// Mitsubishi GX Works2 project: Group555   PLC: FX3G

// global labels: Global1
VAR_GLOBAL
  StartDay AT X007 : BOOL;
  EmergencySwitch AT X011 : BOOL;
  StartLamp AT Y007 : BOOL;
  Yeast_start_register AT D1100 : REAL;
  Malt_start_register AT D1102 : REAL;
  Hops_start_register AT D1104 : REAL;
  Yeast_storage AT D1106 : REAL;
  Malt_storage AT D1108 : REAL;
  Hops_storage AT D1110 : REAL;
  update_storage AT M1 : BOOL;
  Start_cooking AT X001 : BOOL;
  analogInput AT D8280 : INT;
END_VAR
VAR_GLOBAL CONSTANT
  lagerLow : INT;
  PilsnerLow : INT := 2400;
  lager_top : INT := 2000;
  PilsnerTop : INT := 4000;
END_VAR
VAR_GLOBAL
  LagerChoosen AT M2 : BOOL;
  PilsnerChoosen AT M3 : BOOL;
END_VAR
VAR_GLOBAL CONSTANT
  MinYeasteLager : REAL := 150;
  MinMaltLager : REAL := 12;
  MinHopsLager : REAL := 60;
END_VAR
VAR_GLOBAL
  lagerCheackStorage AT M4 : BOOL;
  pilsnerCheackStorage AT M5 : BOOL;
END_VAR
VAR_GLOBAL CONSTANT
  timeLight : INT := 40;
END_VAR
VAR_GLOBAL
  TimerLightTS1 AT TS1 : BOOL;
  light AT Y001 : BOOL;
END_VAR
VAR_GLOBAL CONSTANT
  MinYeastePilsner : REAL := 120;
  MinMaltPilsner : REAL := 6;
  decYeastStorage : REAL := 150;
  decMoltStorage : REAL := 12;
  decHopsStorage : REAL := 60;
  decYeastStorage1 : REAL := 120;
  decMoltStorage1 : REAL := 6;
  decHopsStorage1 : REAL := 53;
END_VAR
VAR_GLOBAL
  Fermentation AT X005 : BOOL;
  FermentationLagerTimer AT TC2 : BOOL;
  TimerFlashLight1 AT TS2 : BOOL;
  light3 AT Y003 : BOOL;
  FermentatioPilnserrTimer AT TC3 : BOOL;
  FermentationLagerOverTimer AT TS2 : BOOL;
  FermentationPlisnerOverTimer AT TS3 : BOOL;
  TimerFermentationOver AT M6 : BOOL;
  Flasing AT X005 : BOOL;
  FlasingFake AT M7 : BOOL;
  FlasingTimer AT TC4 : BOOL;
END_VAR
VAR_GLOBAL CONSTANT
  Flashingtime : INT := 3;
END_VAR
VAR_GLOBAL
  FlashingTimer : INT;
  FlahingTimer AT TC4 : BOOL;
  FlashingLight AT Y003 : BOOL;
  FlashingtOver1 AT TS4 : BOOL;
  FlahingTimer2 AT TC5 : BOOL;
  FlashingtOver2 AT TS5 : BOOL;
  FlashingLight2 AT Y004 : BOOL;
  StartStorage AT X002 : BOOL;
  PackageOneBeer AT X000 : BOOL;
  CountPackage AT D1112 : REAL;
  PackagLight AT Y002 : BOOL;
END_VAR
VAR_GLOBAL CONSTANT
  CounterOfSix : INT := 6;
END_VAR
VAR_GLOBAL
  CounterBottle AT CC1 : BOOL;
  CounteEnd AT CS1 : BOOL;
END_VAR
VAR_GLOBAL CONSTANT
  timeLight2 : INT := 40;
  Add1 : INT := 1;
END_VAR
VAR_GLOBAL
  SumPackage AT D1114 : INT;
  analogOutput AT D8282 : INT;
END_VAR
VAR_GLOBAL CONSTANT
  decimalAmountPackage : INT := 40;  (* . *)
END_VAR
VAR_GLOBAL
  EmptyStorage AT M8 : BOOL;
END_VAR
VAR_GLOBAL CONSTANT
  MinHopsPilsner : REAL := 53;
END_VAR
VAR_GLOBAL
  YeastLagerStorgeOk AT M10 : BOOL;
  MalttLagerStorgeOk AT M11 : BOOL;
  HopsLagerStorgeOk AT M12 : BOOL;
  YeastPilsnerStorgeOk AT M13 : BOOL;
  MalttPilsnerStorgeOk AT M14 : BOOL;
  ExistLagerStorage AT M20 : BOOL;
  ExistPilsnerStorage AT M21 : BOOL;
  HopsPilsnerStorgeOk AT M15 : BOOL;
  EmptyStorageatAtTheStartOfTheDay AT M22 : BOOL;
  StorageLagerCookingOk AT M16 : BOOL;
  StoragePilsnerCookingOk AT M17 : BOOL;
  LagerChoosenHelp AT M40 : BOOL;
  PilsnerChoosenHelp AT M50 : BOOL;
  cookingTimer AT TC1 : BOOL;
END_VAR
VAR_GLOBAL CONSTANT
  ResttPackage : INT;
END_VAR

// task Task_01 (event TRUE, interval 0, priority 31): POU_01

PROGRAM POU_01
(* structured ladder/FBD written out as ST: instructions are called as NAME(EN, inputs, outputs); _pN, _eN, _tN stand for wires *)
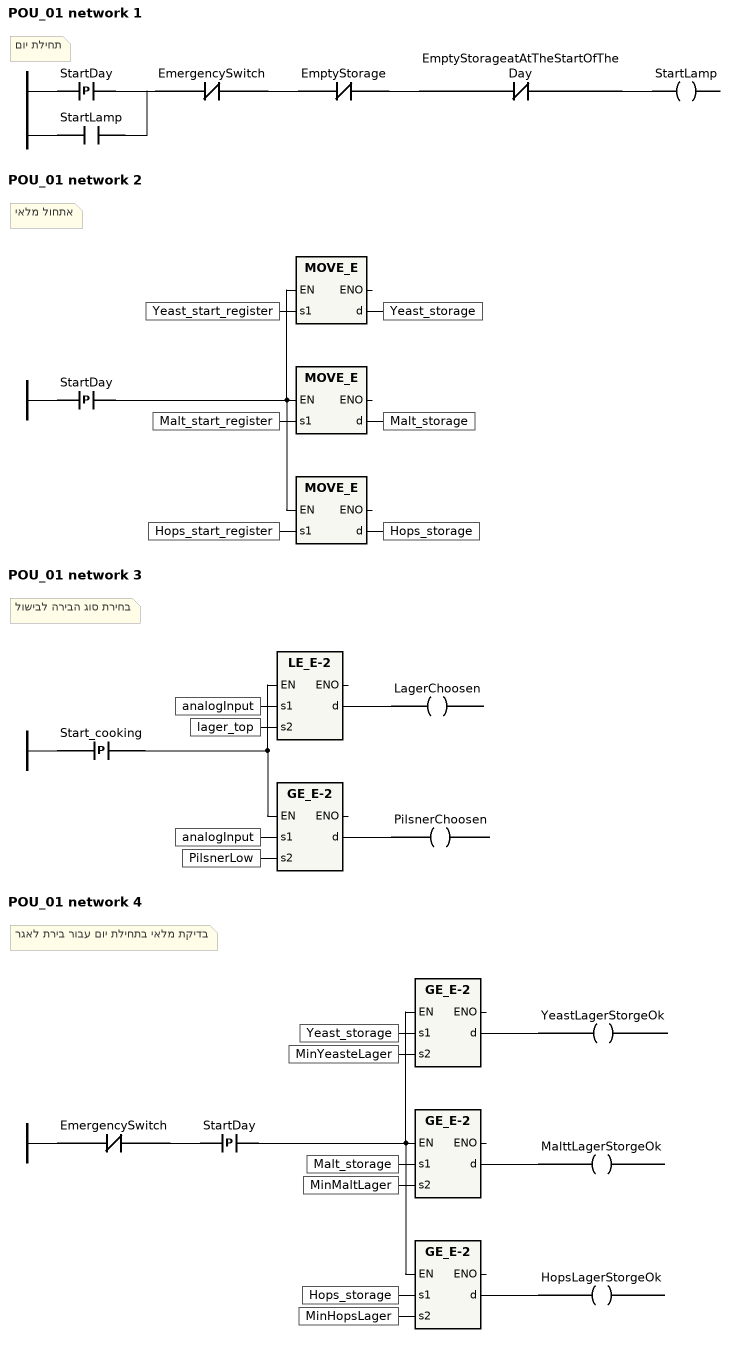
(* network 1 *)
(* תחילת יום *)
StartLamp := (((LDP(TRUE, StartDay) OR StartLamp) AND NOT EmergencySwitch) AND NOT EmptyStorage) AND NOT EmptyStorageatAtTheStartOfTheDay;
(* network 2 *)
(* אתחול מלאי *)
_p1 := LDP(TRUE, StartDay);
MOVE_E(_p1, Yeast_start_register, Yeast_storage);
MOVE_E(_p1, Malt_start_register, Malt_storage);
MOVE_E(_p1, Hops_start_register, Hops_storage);
(* network 3 *)
(* בחירת סוג הבירה לבישול *)
_p1 := LDP(TRUE, Start_cooking);
LE_E(_p1, analogInput, lager_top, _t2);
LagerChoosen := _t2;
GE_E(_p1, analogInput, PilsnerLow, _t3);
PilsnerChoosen := _t3;
(* network 4 *)
(* בדיקת מלאי בתחילת יום עבור בירת לאגר *)
_p1 := NOT EmergencySwitch AND LDP(TRUE, StartDay);
GE_E(_p1, Yeast_storage, MinYeasteLager, _t2);
YeastLagerStorgeOk := _t2;
GE_E(_p1, Malt_storage, MinMaltLager, _t3);
MalttLagerStorgeOk := _t3;
GE_E(_p1, Hops_storage, MinHopsLager, _t4);
HopsLagerStorgeOk := _t4;
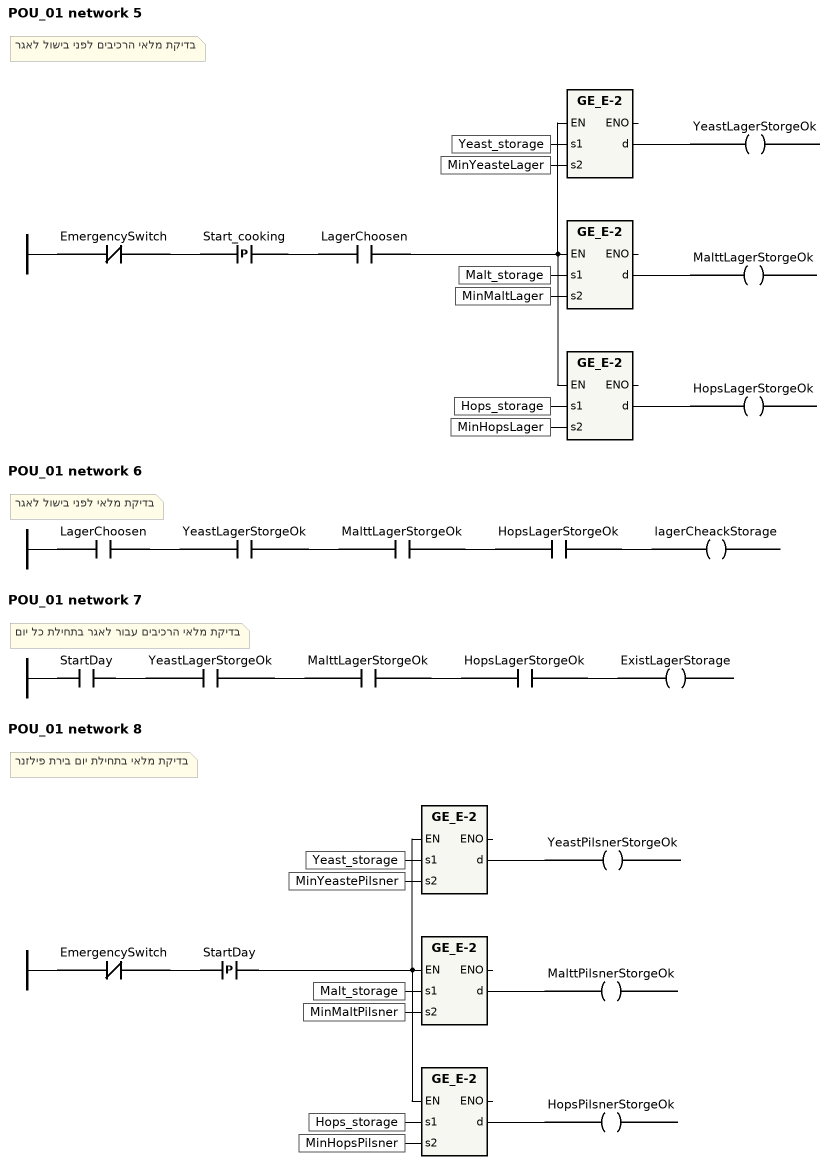
(* network 5 *)
(* בדיקת מלאי הרכיבים לפני בישול לאגר *)
_p1 := NOT EmergencySwitch AND LDP(TRUE, Start_cooking) AND LagerChoosen;
GE_E(_p1, Yeast_storage, MinYeasteLager, _t2);
YeastLagerStorgeOk := _t2;
GE_E(_p1, Malt_storage, MinMaltLager, _t3);
MalttLagerStorgeOk := _t3;
GE_E(_p1, Hops_storage, MinHopsLager, _t4);
HopsLagerStorgeOk := _t4;
(* network 6 *)
(* בדיקת מלאי לפני בישול לאגר *)
lagerCheackStorage := LagerChoosen AND YeastLagerStorgeOk AND MalttLagerStorgeOk AND HopsLagerStorgeOk;
(* network 7 *)
(* בדיקת מלאי הרכיבים עבור לאגר בתחילת כל יום *)
ExistLagerStorage := StartDay AND YeastLagerStorgeOk AND MalttLagerStorgeOk AND HopsLagerStorgeOk;
(* network 8 *)
(* בדיקת מלאי בתחילת יום בירת פילזנר *)
_p1 := NOT EmergencySwitch AND LDP(TRUE, StartDay);
GE_E(_p1, Yeast_storage, MinYeastePilsner, _t2);
YeastPilsnerStorgeOk := _t2;
GE_E(_p1, Malt_storage, MinMaltPilsner, _t3);
MalttPilsnerStorgeOk := _t3;
GE_E(_p1, Hops_storage, MinHopsPilsner, _t4);
HopsPilsnerStorgeOk := _t4;
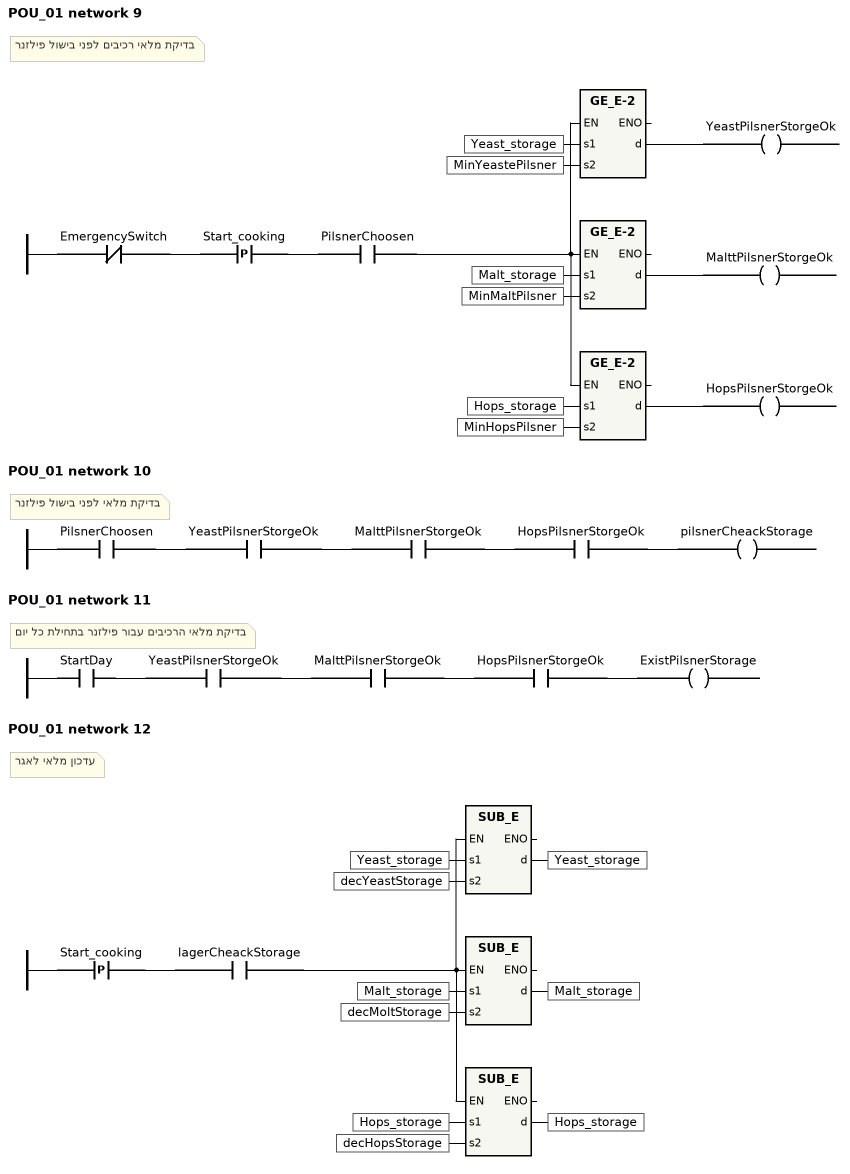
(* network 9 *)
(* בדיקת מלאי רכיבים לפני בישול פילזנר *)
_p1 := NOT EmergencySwitch AND LDP(TRUE, Start_cooking) AND PilsnerChoosen;
GE_E(_p1, Yeast_storage, MinYeastePilsner, _t2);
YeastPilsnerStorgeOk := _t2;
GE_E(_p1, Malt_storage, MinMaltPilsner, _t3);
MalttPilsnerStorgeOk := _t3;
GE_E(_p1, Hops_storage, MinHopsPilsner, _t4);
HopsPilsnerStorgeOk := _t4;
(* network 10 *)
(* בדיקת מלאי לפני בישול פילזנר *)
pilsnerCheackStorage := PilsnerChoosen AND YeastPilsnerStorgeOk AND MalttPilsnerStorgeOk AND HopsPilsnerStorgeOk;
(* network 11 *)
(* בדיקת מלאי הרכיבים עבור פילזנר בתחילת כל יום *)
ExistPilsnerStorage := StartDay AND YeastPilsnerStorgeOk AND MalttPilsnerStorgeOk AND HopsPilsnerStorgeOk;
(* network 12 *)
(* עדכון מלאי לאגר *)
_p1 := LDP(TRUE, Start_cooking) AND lagerCheackStorage;
SUB_E(_p1, Yeast_storage, decYeastStorage, Yeast_storage);
SUB_E(_p1, Malt_storage, decMoltStorage, Malt_storage);
SUB_E(_p1, Hops_storage, decHopsStorage, Hops_storage);
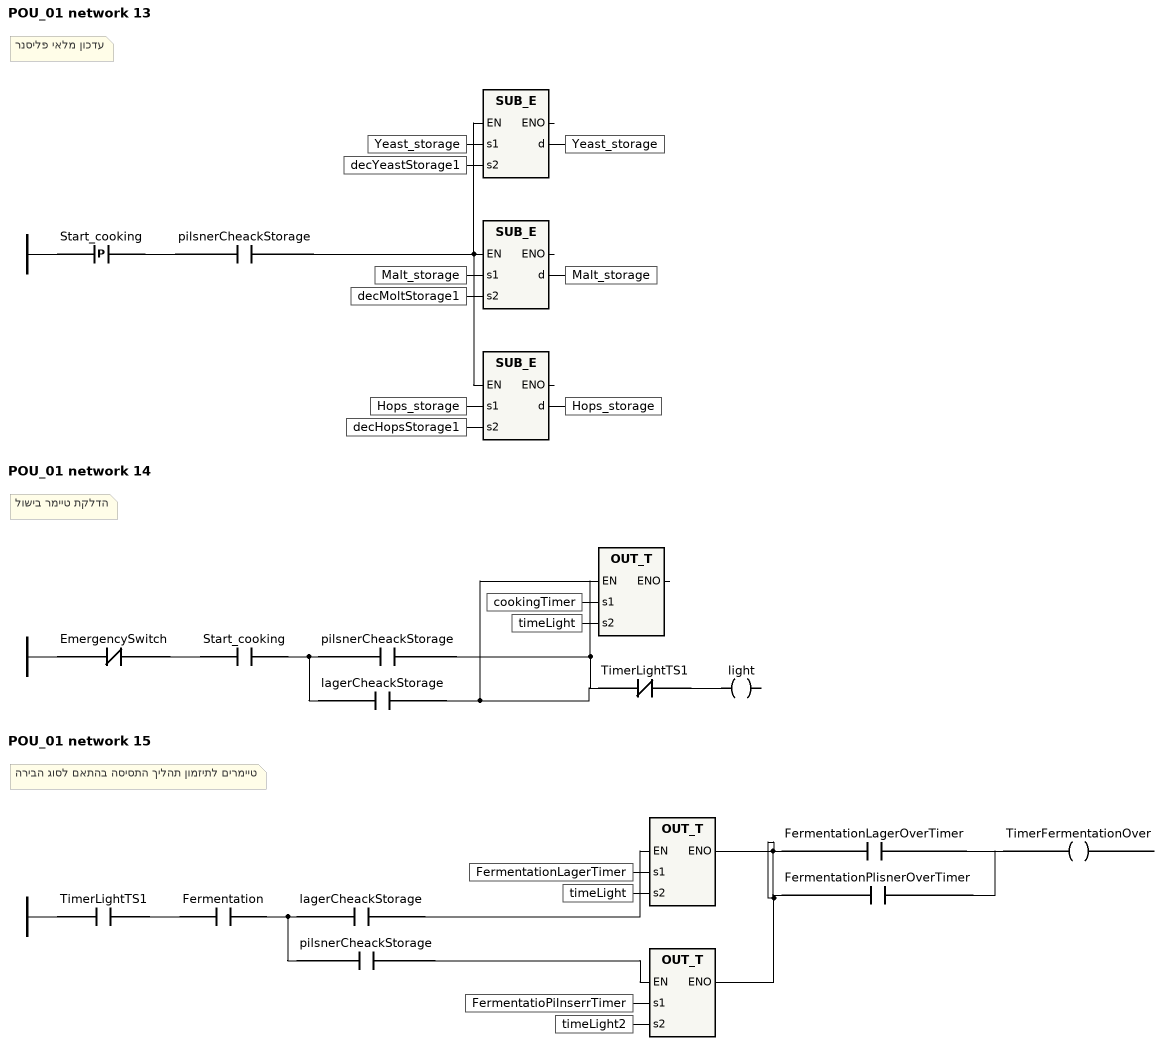
(* network 13 *)
(* עדכון מלאי פליסנר *)
_p1 := LDP(TRUE, Start_cooking) AND pilsnerCheackStorage;
SUB_E(_p1, Yeast_storage, decYeastStorage1, Yeast_storage);
SUB_E(_p1, Malt_storage, decMoltStorage1, Malt_storage);
SUB_E(_p1, Hops_storage, decHopsStorage1, Hops_storage);
(* network 14 *)
(* הדלקת טיימר בישול *)
_p1 := NOT EmergencySwitch AND Start_cooking;
_p2 := (_p1 AND pilsnerCheackStorage) OR (_p1 AND lagerCheackStorage);
OUT_T(_p2, cookingTimer, timeLight);
light := _p2 AND NOT TimerLightTS1;
(* network 15 *)
(* טיימרים לתיזמון תהליך התסיסה בהתאם לסוג הבירה *)
_p1 := TimerLightTS1 AND Fermentation;
_e2 := OUT_T(_p1 AND lagerCheackStorage, FermentationLagerTimer, timeLight);
_e3 := OUT_T(_p1 AND pilsnerCheackStorage, FermentatioPilnserrTimer, timeLight2);
_p4 := _e2 OR _e3;
TimerFermentationOver := (_p4 AND FermentationLagerOverTimer) OR (_p4 AND FermentationPlisnerOverTimer);
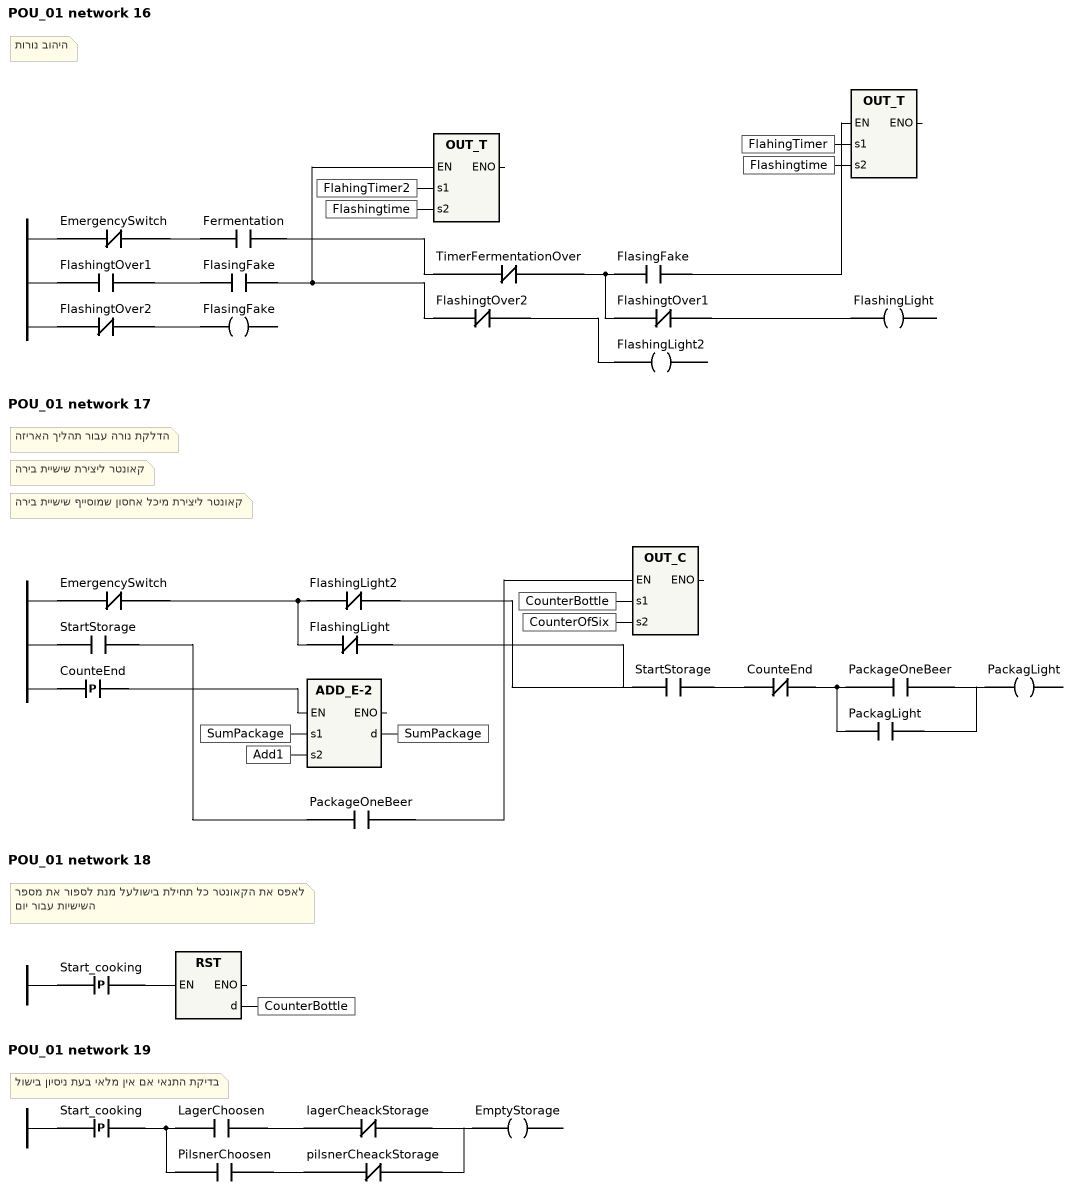
(* network 16 *)
(* היהוב נורות *)
_p1 := NOT EmergencySwitch AND Fermentation AND NOT TimerFermentationOver;
OUT_T(_p1 AND FlasingFake, FlahingTimer, Flashingtime);
FlashingLight := _p1 AND NOT FlashingtOver1;
_p2 := FlashingtOver1 AND FlasingFake;
OUT_T(_p2, FlahingTimer2, Flashingtime);
FlashingLight2 := _p2 AND NOT FlashingtOver2;
FlasingFake := NOT FlashingtOver2;
(* network 17 *)
(* הדלקת נורה עבור תהליך האריזה *)
(* קאונטר ליצירת שישיית בירה *)
(* קאונטר ליצירת מיכל אחסון שמוסייף שישיית בירה *)
_p1 := NOT EmergencySwitch;
_p2 := (((_p1 AND NOT FlashingLight2) OR (_p1 AND NOT FlashingLight)) AND StartStorage) AND NOT CounteEnd;
PackagLight := (_p2 AND PackageOneBeer) OR (_p2 AND PackagLight);
OUT_C(StartStorage AND PackageOneBeer, CounterBottle, CounterOfSix);
ADD_E(LDP(TRUE, CounteEnd), SumPackage, Add1, SumPackage);
(* network 18 *)
(* לאפס את הקאונטר כל תחילת בישולעל מנת לספור את מספר השישיות עבור יום *)
RST(LDP(TRUE, Start_cooking), CounterBottle);
(* network 19 *)
(* בדיקת התנאי אם אין מלאי בעת ניסיון בישול *)
_p1 := LDP(TRUE, Start_cooking);
EmptyStorage := (_p1 AND LagerChoosen AND NOT lagerCheackStorage) OR (_p1 AND PilsnerChoosen AND NOT pilsnerCheackStorage);
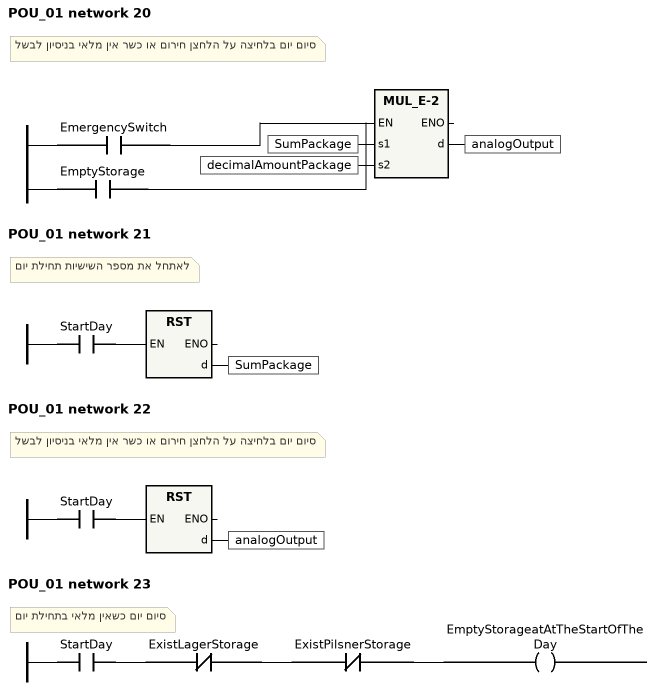
(* network 20 *)
(* סיום יום בלחיצה על הלחצן חירום או כשר אין מלאי בניסיון לבשל *)
MUL_E(EmergencySwitch OR EmptyStorage, SumPackage, decimalAmountPackage, analogOutput);
(* network 21 *)
(* לאתחל את מספר השישיות תחילת יום *)
RST(StartDay, SumPackage);
(* network 22 *)
(* סיום יום בלחיצה על הלחצן חירום או כשר אין מלאי בניסיון לבשל *)
RST(StartDay, analogOutput);
(* network 23 *)
(* סיום יום כשאין מלאי בתחילת יום *)
EmptyStorageatAtTheStartOfTheDay := StartDay AND NOT ExistLagerStorage AND NOT ExistPilsnerStorage;
END_PROGRAM
